FUNCTION F_ComputeEnumSize : UDINT
VAR_INPUT
    anyEnum  : ANY;
END_VAR
VAR
	nTmp : DINT;
END_VAR

IF anyEnum.pValue = NULL OR anyEnum.TypeClass <> __SYSTEM.TYPE_CLASS.TYPE_ENUM THEN
	RETURN;
END_IF

MEMCPY(destAddr:= ADR(nTmp), srcAddr:= anyEnum.pValue, MIN(TO_UDINT(anyEnum.diSize), SIZEOF(nTmp)));
F_ComputeEnumSize := F_ComputeInt32Size(nTmp);

END_FUNCTION

(* stored: Version 1.1.0.1
   POU F_ComputeEnumSize: Id {fed8b217-7dd0-4101-8158-a06e03aee7a9}, SpecialFunc None *)
